FUNCTION_BLOCK FB_Component_SingleValveGuarded IMPLEMENTS I_Component
VAR_INPUT
	sName			: STRING[50];
	tTimeout		: TIME := T#0S;
END_VAR

VAR_IN_OUT
	bSensExtended	: BOOL;
	bSensRetracted	: BOOL;
	bOutput			: BOOL;
END_VAR

VAR_OUTPUT
	bEnabled     	: BOOL;
	eState			: E_State := E_State.DISABLED;
	eNextState		: E_State := E_State.DISABLED;
	sStatusText 	: STRING[100];
	
	bIsExtended		: BOOL;
	bIsRetracted	: BOOL;
END_VAR

VAR
	bRetracting		: BOOL;
	bExtending		: BOOL;
	tTimeoutTimer	: TON;

	eLastState		: E_State;
	
	Components		: ARRAY [0..2] OF I_Component;
	
	fbPiston		: FB_Component_SingleValve;
	fbReedExtended	: FB_Component_ReedSwitch;
	fbReedRetracted	: FB_Component_ReedSwitch;
END_VAR

VAR CONSTANT
	DISABLED		: E_State := E_State.DISABLED;
	READY			: E_State := E_State.READY;
	BUSY			: E_State := E_State.BUSY;
	DONE			: E_State := E_State.DONE;
	HALTED			: E_State := E_State.HALTED;
	TIMEOUT			: E_State := E_State.TIMEOUT;
END_VAR

tTimeoutTimer(PT := tTimeout);

fbPiston(sName := '', tTimeout 	:= T#0S, bOutput := bOutput);
fbReedExtended(sName := '', bRawSignal 	:= bSensExtended, tTimeout := T#0S);
fbReedRetracted(sName := '', bRawSignal 	:= bSensRetracted, tTimeout := T#0S);

Components[0] := fbPiston;
Components[1] := fbReedExtended;
Components[2] := fbReedRetracted;

bIsExtended		:= fbReedExtended.bSensorActive;
bIsRetracted	:= fbReedRetracted.bSensorActive;

eState := eNextState;

CASE eState OF
	DISABLED: 	sStatusText := 'piston disabled';
	READY: 		sStatusText :=  CONCAT(CONCAT(SEL(bIsExtended = TRUE, '', 'piston extended and '),SEL(bIsRetracted = TRUE, '', 'piston retracted and ')), 'ready to operate');
	
	BUSY: 		IF bExtending THEN
					sStatusText := 'piston extending';
					IF fbReedExtended.bSensorActive THEN
						eNextState := TIMEOUT;
					ELSE
						fbPiston.M_Extend();
					END_IF
				END_IF
				IF bRetracting THEN
					sStatusText := 'piston retracting';
					IF fbReedRetracted.bSensorActive THEN
						eNextState := TIMEOUT;
					ELSE
						fbPiston.M_Retract();
					END_IF
				END_IF
			
	TIMEOUT:	sStatusText := 'piston in timeout';
				bExtending  := FALSE;
				bRetracting := FALSE;
				tTimeoutTimer(IN := TRUE);
				
				IF tTimeoutTimer.Q THEN
					tTimeoutTimer(IN := FALSE);
					eNextState := READY;
				END_IF
				
	HALTED:		sStatusText := 'piston halted';
END_CASE

{warning 'add method implementation '}
METHOD M_Disable : BOOL
VAR
	idx	: INT := 0;
END_VAR
IF eState = READY THEN
	bEnabled	:= FALSE;
	eNextState	:= DISABLED;
	
	FOR idx := 0 TO 2 DO
    	Components[idx].M_Disable();
	END_FOR;
END_IF
END_METHOD

{warning 'add method implementation '}
METHOD M_Enable : BOOL

VAR
	idx: INT;
END_VAR
IF eState = DISABLED THEN
	bEnabled	:= TRUE;
	eNextState	:= READY;
	
	FOR idx := 0 TO 2 DO
    	Components[idx].M_Enable();
	END_FOR;
END_IF
END_METHOD

METHOD M_Extend : BOOL
VAR_INPUT
END_VAR
IF eState = READY AND NOT fbReedExtended.bSensorActive THEN
	bExtending 	:= TRUE;
	eNextState	:= BUSY;
END_IF
END_METHOD

{warning 'add method implementation '}
METHOD M_Halt : BOOL

VAR
	idx: INT;
END_VAR
IF eState <> HALTED AND eState <> DISABLED THEN
	eLastState 		:= eState;
	eNextState		:= HALTED;
	FOR idx := 0 TO 2 DO
		Components[idx].M_Halt();
	END_FOR;
END_IF
END_METHOD

{warning 'add method implementation '}
METHOD M_Resume : BOOL

VAR
	idx: INT;
END_VAR
IF eState = HALTED THEN
	eNextState := eLastState;
	FOR idx := 0 TO 2 DO
		Components[idx].M_Resume();
	END_FOR;
END_IF
END_METHOD

METHOD M_Retract : BOOL
VAR_INPUT
END_VAR
IF eState = READY AND NOT fbReedRetracted.bSensorActive  THEN
	bRetracting	:= TRUE;
	eNextState	:= BUSY;
END_IF
END_METHOD

END_FUNCTION_BLOCK

(* stored: Version 1.1.0.1, ProductVersion 3.1.4024.15
   POU FB_Component_SingleValveGuarded: Id {62ac951b-123f-4803-bb89-42aab24e981e}, SpecialFunc None
   Method M_Disable: Id {c6b4994e-a0da-440e-9ca1-3cf41ca8d7bf}
   Method M_Enable: Id {e1ec62f0-3e96-4b93-9f77-720e89ed850a}
   Method M_Extend: Id {7b5b372b-00b9-4b2c-b2c5-99e037e088b9}
   Method M_Halt: Id {11a97c53-cc9e-4a78-a566-da9303d32528}
   Method M_Resume: Id {7dae0265-d6b8-4712-ba2c-690c76d5615a}
   Method M_Retract: Id {e8c004e6-1cb6-4652-a159-4035bb0a34cc} *)
